INTERFACE I_Mode

METHOD Auto
VAR_INPUT
	bEnable : BOOL;
END_VAR
END_METHOD

METHOD Manual
VAR_INPUT
	bEnable : BOOL;
END_VAR
END_METHOD

METHOD OFF 
VAR_INPUT
	bEnable : BOOL;
END_VAR
END_METHOD

END_INTERFACE

(* stored: Version 1.1.0.1, ProductVersion 3.1.4024.12
   Itf I_Mode: Id {52df050c-22df-43bf-aacb-4bbb8d640659}
   Method Auto: Id {0c89b980-bbec-4646-80f1-38627076a9bc}
   Method Manual: Id {646cefd6-055d-473d-a7ff-0335cc1fc8cc}
   Method OFF: Id {fb413af2-9ed3-4835-80cd-e4fa7eedafeb} *)
